Yaskawa INFORM job: TEST-ODW-R2.JBI

/JOB
//NAME TEST-ODW-R2
///FOLDERNAME INNE
//POS
///NPOS 1,1,1,0,0,0
///TOOL 0
///POSTYPE PULSE
///PULSE
C00000=169402,152846,102070,-9296,84238,-70965
BC00000=248646,1341745,985433
EC00000=0,0
//INST
///DATE 2023/11/01 18:40
///ATTR SC,RW
///GROUP1 RB1,BS1
///GROUP2 ST1
NOP
'test-odw-r2
MOVJ C00000 BC00000 VJ=100.00  +MOVJ EC00000 VJ=100.00
END
